VAR_GLOBAL PERSISTENT
	PersMachPar					: ST_MachPar;
	PersSysPar					: ST_SysPar;
END_VAR
VAR_GLOBAL CONSTANT
	MAX_ZONES					: INT:= 7;
END_VAR

(* stored: Version 1.1.0.1, ProductVersion 3.1.4020.12
   GVL GVL: Id {a030a360-f43d-49e5-918f-501fc58fede1} *)
